TYPE ST_FB_MGMT_Stellwert :
STRUCT
	Betrieb		: BOOL;

(*Heizung*)
	BHKW1_Anforderung       			: BOOL;
 	BHKW2_Anforderung       			: BOOL;
 	BWT_Anforderung       				: BOOL;
 	PWT1_Anforderung       				: BOOL;
 	AKM_Anforderung       				: BOOL;

(*Freigabe_Entziehung*)
	BHKW1_Freigabe_Entziehung            : BOOL;
	BHKW2_Freigabe_Entziehung            : BOOL;
	BWT_Freigabe_Entziehung             : BOOL;
	PWT1_Freigabe_Entziehung            : BOOL;
	WP_Freigabe_Entziehung              : BOOL;

(*Kuehlung*)
	gruennetz_Kuehlung_Anforderung      : BOOL;
    Kuehlung_KKKW_Anforderung        	: BOOL;

(*Kuehlung/Heitung*)
	Waermepumpe_945_Anforderung       	: BOOL;

(*Speicher*)
	Anford_Kuehlwasser				: BOOL;
	Anford_Kuehlwarmwasser			: BOOL;
	Anford_Kuehlkaltwasser			: BOOL;
	blaunetz_Kuehlung_Anforderung	: BOOL;



END_STRUCT
END_TYPE

(* stored: Version 1.1.0.1, ProductVersion 3.1.4024.9
   DUT ST_FB_MGMT_Stellwert: Id {42190553-6229-4a97-af2a-b8e4aaefc75a} *)
